(* PLC project Unnamed, Unknown Unnamed 1 *)
(* stored: creationDateTime 2022-09-05T09:02:48, modificationDateTime 2022-09-20T11:48:55 *)

PROGRAM program0
  VAR
    LocalVar0 : DINT;
    LocalVar1 : DINT;
  END_VAR

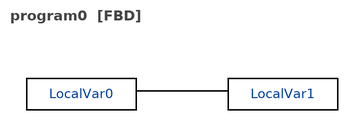
(* FBD diagram, written out as Structured Text *)
LocalVar1 := LocalVar0;
END_PROGRAM

CONFIGURATION config
  RESOURCE resource1 ON PLC
    TASK task0(INTERVAL := T#20ms, PRIORITY := 0);
    PROGRAM instance0 WITH task0 : program0;
  END_RESOURCE
END_CONFIGURATION
